// TIA Portal V16 export
// export: Created 2024-08-19T08:04:44.0785637Z, ExportSetting WithDefaults, DisplayName Totally Integrated Automation Portal, DisplayVersion V16, DisplayName TIA Portal Version Control Interface, DisplayVersion V16, DisplayName TIA Portal Openness, DisplayVersion V16, DisplayName STEP 7 Professional, DisplayVersion V16, DisplayName STEP 7 Safety, DisplayVersion V16, DisplayName WinCC Professional, DisplayVersion V16
TYPE "UT00851_Sy_ConstAiScaleData"
TITLE = Static UDT [SYSTEM CONSTANTS] — Analog Input Scale Data and Ranges
// PRACTICAL SERIES AUTOMATION LIBRARY (PAL)   —   COPYRIGHT 2020 – M. GLEDHILL (MIT LICENCE)
//                   ———— ◆ ————
// FULL ONLINE DOCUMENTATION IS AVAILABLE AT: https://practicalseries.com/2001-pal/index.html
// stored: IsFailsafeCompliant false
   STRUCT
      revInfo { ExternalWritable := 'False'} : "UT01000_St_SysRevision";   // ▀▀▀▀ UDT CURRENT REVISION
      ___________0010_0 { ExternalAccessible := 'False'; ExternalVisible := 'False'; ExternalWritable := 'False'} : Bool;
      ___________0010_1 { ExternalAccessible := 'False'; ExternalVisible := 'False'; ExternalWritable := 'False'} : Bool;   // ▀▀▀▀ AI DEVICE ID
      AI_TAG { ExternalWritable := 'False'} : String[20] := 'AAAnnn';   // Device or instrument tag
      ___________0020_0 { ExternalAccessible := 'False'; ExternalVisible := 'False'; ExternalWritable := 'False'} : Bool := false;
      ___________0020_1 { ExternalAccessible := 'False'; ExternalVisible := 'False'; ExternalWritable := 'False'} : Bool;   // ▀▀▀▀ AI SCALED RANGE DATA
      SCALE_MIN { ExternalWritable := 'False'} : Real := 0.0;   // Minimum value of the scaled signal
      SCALE_MAX { ExternalWritable := 'False'} : Real := 100.0;   // Maximum value of the scaled signal
      SCALE_UNITS { ExternalWritable := 'False'} : String[20] := '%';   // Scaled signal engineering units
      SCALE_DESC { ExternalWritable := 'False'} : String[60] := 'Default range 0.0-100.0%';   // Scaled signal type information (plain English)
      ___________0030_0 { ExternalAccessible := 'False'; ExternalVisible := 'False'; ExternalWritable := 'False'} : Bool := false;
      ___________0030_1 { ExternalAccessible := 'False'; ExternalVisible := 'False'; ExternalWritable := 'False'} : Bool;   // ▀▀▀▀ AI OUT OF RANGE DATA
      LIMIT_UNDER { ExternalWritable := 'False'} : Real := 0.0;   // Lower limit of scaled signal before under-range (in engineering uints)
      LIMIT_OVER { ExternalWritable := 'False'} : Real := 100.0;   // Upper limit of scaled signal before over-range (in engineering uints)
      ___________0040_0 { ExternalAccessible := 'False'; ExternalVisible := 'False'; ExternalWritable := 'False'} : Bool := false;
      ___________0040_1 { ExternalAccessible := 'False'; ExternalVisible := 'False'; ExternalWritable := 'False'} : Bool;   // ▀▀▀▀ AI USER INFORMATION
      USER_INFO_1 : String[60] := 'Optional user information';   // Optional user information (text) line 1
      USER_INFO_2 : String[60] := 'Optional user information';   // Optional user information (text) line 2
      USER_INFO_3 : String[60] := 'Optional user information';   // Optional user information (text) line 3
      USER_INFO_4 : String[60] := 'Optional user information';   // Optional user information (text) line 4
      USER_INFO_5 : String[60] := 'Optional user information';   // Optional user information (text) line 5
   END_STRUCT;
   // revInfo.REV_BLOCK := 'UT00851';
   // revInfo.REV_NUMBER := '001.000';
   // revInfo.REV_DATE := '2024-05-11';
   // revInfo.REV_AUTHOR := 'M. Gledhill';
END_TYPE
